// TIA Portal V19 export
DATA_BLOCK "Settings"   // DB6
{ DB_Accessible_From_OPC_UA := 'FALSE' }
// stored: DBAccessibleFromOPCUA false, DBAccessibleFromWebserver false, MemoryReserve 100
   VAR
      diagPlc : "LAF_typePlcDiag";   // HMI interface PLC diag / HMI Schnittstelle PLC Diagnose
      checksum : "LAF_typeChecksum";   // HMI interface PLCChecksum / HMI Schnittstelle PLCChecksum
      diagMemCard : "LAF_typeMemCardDiag";   // HMI interface SMCDiag / HMI Schnittstelle SMCDiag
      cycleTimes : "LAF_typeGlobalRuntime";
      setLocalPlcTime : "LAF_typeSetPlcTime";
      ITConnection : Bool := FALSE;   // Provides a visual representation of the connection with the IT systems.
   END_VAR
BEGIN
END_DATA_BLOCK
